FUNCTION_BLOCK ARRAY2ARRAY_2_LREAL
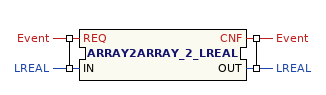
  EVENT_INPUT
    REQ WITH IN;
  END_EVENT
  EVENT_OUTPUT
    CNF WITH OUT;
  END_EVENT
  VAR_INPUT
    IN : LREAL;
  END_VAR
  VAR_OUTPUT
    OUT : LREAL;
  END_VAR
END_FUNCTION_BLOCK
